{attribute 'qualified_only'}
VAR_GLOBAL		
	B1: BOOL; 	// Endschalter Links
	B2: BOOL;	// Endschalter Rechts
	F1: BOOL;	// Thermorelais
	S1: BOOL;	// Taster Start
	S2: BOOL;	// Taster NotHalt
	S3: BOOL;	// Taster Reset
END_VAR

(* stored: Version 1.1.0.1, ProductVersion 3.1.4024.4
   GVL SimDI: Id {c2d05302-d374-4f85-80dd-41006a3e3277} *)
